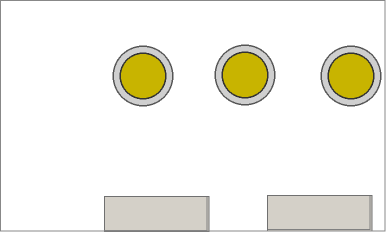
VISUALIZATION Visualization  // 386x232
    Lamp1 (108,41 70x70), variable: I0.bLampeGruen, style: Lamp-Lamp1-Yellow
    Lamp1 (210,40 70x70), variable: I0.bLampeGelb, style: Lamp-Lamp1-Yellow
    Lamp1 (316,41 70x70), variable: I0.bLampeRot, style: Lamp-Lamp1-Yellow
    Button (104,196 105x36)
        tap I0.bSchalterBlau
    Button (267,195 105x36)
        tap I0.bSchalterGelb
END_VISUALIZATION

(* stored: Version 1.1.0.1, ProductVersion 3.1.4024.12
   Visu Visualization: Id {8fbb9241-99eb-4d7c-95bb-fc4d61705eb9} *)
